// TIA Portal V19 export
TYPE "ITF_A01"
// stored: Access Published
   STRUCT
      AreaInterface : "AreaInterface";
      CoilHandling_MachineInterface { S7_SetPoint := 'True'} : "MachineInterface";
      Infeed_REQ_ON : Bool := FALSE;
      PB : Struct
         MB1_PB_Reset : Bool := FALSE;
         LB114_Interlock_PB_FeedA02 : Bool;
         Area_DataOut_LampCycle : Bool;
      END_STRUCT;
      Safety_SuperUser : Struct
         PbSafetyReset : Bool;
         SgnSafetyReset : Bool;
      END_STRUCT;
      Safety_EntryEnable : Struct
         Z01 : Bool;
         Z02 : Bool;
         Z03 : Bool;
         Z05 : Bool;
         Z10 : Bool;
      END_STRUCT;
      Safety_CtrlSafe : Struct
         HU_Decoilers_Motor : Bool;
         HU_Decoilers_StandbyValve : Bool;
         HU_Decoilers_SafetyValve_HorizRot : Bool;
         HU_Decoilers_SafetyValve_Decoiler1 : Bool;
         HU_Decoilers_SafetyValve_Decoiler2 : Bool;
         HU_A01_Motor : Bool;
         HU_A01_StandbyValve : Bool;
         HU_A01_DegasValve : Bool;
         HU_A01_SafetyValve_CoilCar : Bool;
         HU_A01_SafetyValve_Peeler : Bool;
         HU_A01_SafetyValve_JB_CutRest : Bool;
         HU_A01_SafetyValve_JB_CutWork : Bool;
         Sinamics_CoilCar : Bool;
         Sinamics_DecoilersTranslation : Bool;
         Sinamics_Decoiler1 : Bool;
         Sinamics_Decoiler2 : Bool;
         Sinamics_Straightener : Bool;
         Sinamics_JB_Torch : Bool;
         Sinamics_JB_PinchR : Bool;
      END_STRUCT;
      Doors_Closed { ExternalWritable := 'False'} : Bool;
      Production_Running : Bool;
      Production_Halted : Struct
         Code : Int;
         Message_N { ExternalWritable := 'False'} : Int;
      END_STRUCT;
      MaterialCounter : "MatCountData";   // = "CoilHandlingMatCounter_PERS".PersistentValues.Data.CounterValue
      MaterialPresence { ExternalAccessible := 'False'; ExternalVisible := 'False'; ExternalWritable := 'False'} : Bool := TRUE;
      MaterialPresence_StraightenerEntry { ExternalAccessible := 'False'; ExternalVisible := 'False'; ExternalWritable := 'False'} : Bool := TRUE;
      MaterialPresence_StraightenerExit { ExternalAccessible := 'False'; ExternalVisible := 'False'; ExternalWritable := 'False'} : Bool := TRUE;
      MaterialPresence_JBPinchExit { ExternalAccessible := 'False'; ExternalVisible := 'False'; ExternalWritable := 'False'} : Bool := TRUE;
      Material_STS : Int;
      Decoiler_InLine : Int;
      Coil_Diameter : Real;
      WeldDone : Bool;
      Deroga_Spessore_Errato : Bool;
      Spessore_Lamiera_Errato : Bool;
      Spessore_Lamiera_Errore_Valore : Real;
      Spessore_Lamiera_Sensore_Valore : Real;
      Provino_Eseguito : Bool;
      Loop1_COut { S7_SetPoint := 'True'} : "SmartLoopControl_COut";
      Loop1_Lamp { S7_SetPoint := 'True'} : Bool;
      Loop1_MachineInterface { S7_SetPoint := 'True'} : "MachineInterface";
      NxtEndOfMaterial { S7_SetPoint := 'True'} : Bool;
      EmptyingConfirmed : Bool;
      StraightnerPowerOn : Bool;
      FreeBool : Array[1..16] of Bool;
      FreeLReal : Array[1..16] of LReal;
      FreeDINT : Array[1..16] of DInt;
   END_STRUCT;
END_TYPE
